(*

.. <legal notes>

legal notes
=================
| SPDX-FileCopyrightText: © 2026 Oleksandr Tiutyk <trofimich@gmail.com>
| SPDX-License-Identifier: LGPL-3.0-only
| For details check: LGPL-3.0-only_

.. _LGPL-3.0-only: https://www.gnu.org/licenses/lgpl-3.0.en.html

.. </legal notes>

*)

FUNCTION_BLOCK ABSTRACT InputOutputDevice EXTENDS SimpleDevice IMPLEMENTS IInputDevice, IOutputDevice

METHOD PROTECTED ABSTRACT OnProcessInput
END_METHOD

METHOD PROTECTED ABSTRACT OnProcessOutput
END_METHOD

METHOD FINAL ProcessInput
VAR
	exceptionCode : __SYSTEM.ExceptionCode;
	exception : Core.IException;
	severity : Core.ERROR_SEVERITY;
END_VAR
__TRY
	OnProcessInput();
__CATCH(exceptionCode)	
	exception := Core.ExceptionManager.GetLastException(exceptionCode);
					
	severity := _ExceptionSeverityResolver.GetSeverity(exception, __POUNAME());

	SetException(exception, severity);	
__ENDTRY
END_METHOD

METHOD FINAL ProcessOutput
VAR
	exceptionCode : __SYSTEM.ExceptionCode;
	exception : Core.IException;
	severity : Core.ERROR_SEVERITY;
END_VAR
__TRY
	OnProcessOutput();
__CATCH(exceptionCode)	
	exception := Core.ExceptionManager.GetLastException(exceptionCode);
					
	severity := _ExceptionSeverityResolver.GetSeverity(exception, __POUNAME());

	SetException(exception, severity);	
__ENDTRY
END_METHOD

END_FUNCTION_BLOCK

(* stored: Version 1.1.0.1
   POU InputOutputDevice: Id {d3cfaf06-a014-47b7-8cf6-98a0cc083f94}, SpecialFunc None
   Folder Methods to override: Id {c65c0bbf-e1ef-43ca-a18f-3c425c65c3bc}
   Method OnProcessInput: Id {94e71efd-bb71-4095-9cb0-5f4f8a38c0d8}
   Method OnProcessOutput: Id {6751103a-6dfb-417d-8b22-87cbdffa3af8}
   Method ProcessInput: Id {253f2967-16b7-4926-8948-e00e6a6f87fb}
   Method ProcessOutput: Id {41595c71-5414-4593-a797-cb95863046c3} *)
